{attribute 'GeneratedUsingTerminal: EPP1111-0000-0016'}
{attribute addProperty BoxType "EPP1111-0000-0016"}
{attribute addProperty Id "EtcSlaveTerminalBaseID_InputsAT %I*ID_Inputs_07C9D28F2WcStateAT %I*WcState_9091E0EB2InfoDataAT %I*InfoData_32EB74EA10"}
{attribute addProperty CRC "585421493"}
{attribute addProperty Size "14"}
TYPE EPP1111_22E4D2B5 EXTENDS EtcSlaveTerminalBase :
STRUCT
	{attribute addProperty Name "ID_Inputs"}
	ID_Inputs : ID_Inputs_07C9D28F;
	{attribute addProperty Name "WcState"}
	WcState : WcState_9091E0EB;
	{attribute addProperty Name "InfoData"}
	InfoData : InfoData_32EB74EA;
END_STRUCT
END_TYPE

(* stored: Version 1.2.0.0, ProductVersion 3.1.4024.9
   DUT EPP1111_22E4D2B5: Id {87a1cbc5-ca67-4771-b603-37d63001c7e5} *)
